INTERFACE I_JsonResponseBuilder EXTENDS I_ResponseBuilder

METHOD PUBLIC CopyJsonDocument : UDINT
VAR_INPUT
	pString : POINTER TO STRING;
	Size : UDINT;
END_VAR
END_METHOD

METHOD PUBLIC GetJsonDocument : T_MAXSTRING
VAR_INPUT
END_VAR
END_METHOD

METHOD PUBLIC GetJsonDocumentLength : UDINT
VAR_INPUT
END_VAR
END_METHOD

METHOD PUBLIC ResetDocument
VAR_INPUT
END_VAR
END_METHOD

END_INTERFACE

(* stored: Version 1.1.0.1, ProductVersion 3.1.4024.12
   Itf I_JsonResponseBuilder: Id {35125eb8-87c9-0126-04de-a2940cb152de}
   Method CopyJsonDocument: Id {0dc04f0a-6081-08c3-3a21-9420297de638}
   Method GetJsonDocument: Id {3d8eb2c5-d2e0-0444-39f0-ed668c2dab0b}
   Method GetJsonDocumentLength: Id {f9095613-93ed-05db-35ad-079c3ed56b28}
   Method ResetDocument: Id {9f156676-272d-0047-38e6-4ac6651ef141} *)
